// ---- VISUs/StepBlockDetection.TcVIS
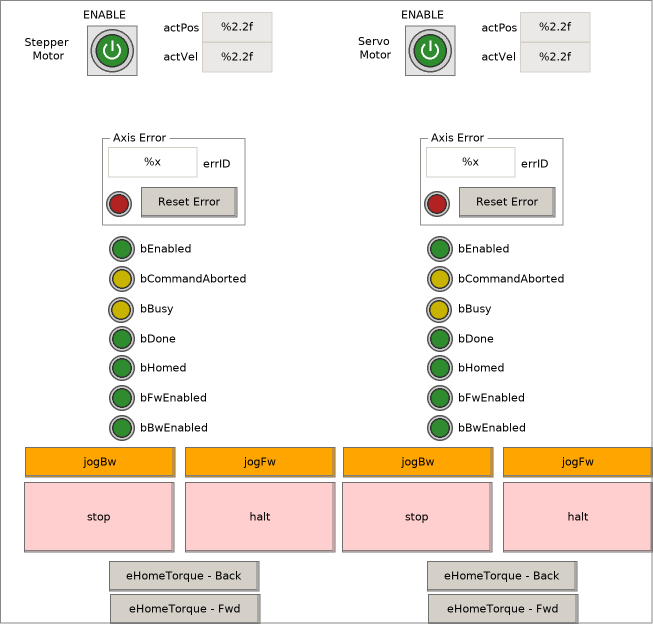
VISUALIZATION StepBlockDetection  // 653x624
    GroupBox (102,130 143x95), "Axis Error"
    Lamp1 (104,189 30x30), variable: GVL.astAxes[1].stStatus.bError, style: Lamp-Lamp1-Red
    Button (141,187 96x30), "Reset Error", pressed state: GVL.astAxes[3].stControl.bReset, text list: 'languageTable', text index: "reset"
        OnMouseClick: toggle GVL.astAxes[1].stControl.bReset
    Textfield (108,147 89x30), "%x", text variable: GVL.astAxes[1].stStatus.nErrorID
    Textfield (200,149 44x30), "errID", text list: 'languageTable', text index: "errID"
    Textfield (137,413 117x30), "bBwEnabled", text list: 'languageTable', text index: "bBwEnabled"
    Lamp1 (107,234 30x30), variable: GVL.astAxes[1].stStatus.bEnabled, style: Lamp-Lamp1-Green
    Textfield (137,234 117x30), "bEnabled", text list: 'languageTable', text index: "bEnabled"
    Lamp1 (107,264 30x30), variable: GVL.astAxes[1].stStatus.bCommandAborted, style: Lamp-Lamp1-Yellow
    Textfield (137,264 117x30), "bCommandAborted", text list: 'languageTable', text index: "bCommandAborted"
    Textfield (137,294 117x30), "bBusy", text list: 'languageTable', text index: "bBusy"
    Lamp1 (107,324 30x30), variable: GVL.astAxes[1].stStatus.bDone, style: Lamp-Lamp1-Green
    Textfield (137,324 117x30), "bDone", text list: 'languageTable', text index: "bDone"
    Lamp1 (107,353 30x30), variable: GVL.astAxes[1].stStatus.bHomed, style: Lamp-Lamp1-Green
    Textfield (137,353 117x30), "bHomed", text list: 'languageTable', text index: "bHomed"
    Lamp1 (107,383 30x30), variable: GVL.astAxes[1].stStatus.bFwEnabled AND NOT GVL.astAxes[1].stStatus.bInterlockedFwd, style: Lamp-Lamp1-Green
    Lamp1 (107,413 30x30), variable: GVL.astAxes[1].stStatus.bBwEnabled AND NOT GVL.astAxes[1].stStatus.bInterlockedBwd, style: Lamp-Lamp1-Green
    Textfield (137,383 117x30), "bFwEnabled", text list: 'languageTable', text index: "bFwEnabled"
    Lamp1 (106,295 30x30), variable: GVL.astAxes[1].stStatus.bBusy, style: Lamp-Lamp1-Yellow
    Textfield (202,12 70x30), "%2.2f", text variable: GVL.astAxes[1].stStatus.fActPosition
    Textfield (148,13 54x30), "actPos", text list: 'languageTable', text index: "actposition"
    Textfield (152,42 49x30), "actVel", text list: 'languageTable', text index: "actVelocity"
    Textfield (202,42 70x30), "%2.2f", text variable: GVL.astAxes[1].stStatus.fActVelocity
    Textfield (80,2 92x26), "ENABLE", text list: 'languageSupport', text index: "enable"
    PowerSwitch (87,24 50x53), variable: GVL.astAxes[1].stControl.bEnable, behaviour: TOGGLE, style: Switch-PowerSwitch-Green
    Button (25,447 150x30), "jogBw", text list: "languageSupport", text index: "jogBw"
        OnMouseDown: execute { GVL.astAxes[1].stControl.eCommand:=E_MotionFunctions.eJog; GVL.astAxes[1].stControl.bJogBwd:= TRUE; }
        OnMouseClick: execute {  }
        OnMouseUp: execute { GVL.astAxes[1].stControl.bJogBwd:= FALSE; }
    Button (185,447 150x30), "jogFw", text list: "languageSupport", text index: "jogFw"
        OnMouseDown: execute { GVL.astAxes[1].stControl.eCommand:=E_MotionFunctions.eJog; GVL.astAxes[1].stControl.bJogFwd:= TRUE; }
        OnMouseClick: execute {  }
        OnMouseUp: execute { GVL.astAxes[1].stControl.bJogFwd:= FALSE; }
    Button (185,482 150x70), "halt", pressed state: GVL.astAxes[1].stControl.bHalt, input disabled if: GVL.astAxes[1].stStatus.bGeared, text list: "languageSupport", text index: "halt"
        toggle GVL.astAxes[1].stControl.bHalt
    Button (24,482 150x70), "stop", pressed state: GVL.astAxes[1].stControl.bStop, input disabled if: GVL.astAxes[1].stStatus.bGeared, text list: "languageSupport", text index: "stop"
        toggle GVL.astAxes[1].stControl.bStop
    Button (109,561 150x30), "eHomeTorque - Back", input disabled if: GVL.astAxes[1].stStatus.bGeared
        OnMouseClick: execute {
            GVL.astAxes[1].stControl.eCommand:=E_MotionFunctions.eHome;
            GVL.astAxes[1].stConfig.eHomeSeq:=E_HomingRoutines.eHomeToBlock_Bwd;
            GVL.astAxes[1].stControl.bExecute:=TRUE;
        }
    Button (110,594 150x30), "eHomeTorque - Fwd", input disabled if: GVL.astAxes[3].stStatus.bGeared
        OnMouseClick: execute {
            GVL.astAxes[1].stControl.eCommand:=E_MotionFunctions.eHome;
            GVL.astAxes[1].stConfig.eHomeSeq:=E_HomingRoutines.eHomeToBlock_Fwd;
            GVL.astAxes[1].stControl.bExecute:=TRUE;
        }
    GroupBox (420,130 143x95), "Axis Error"
    Lamp1 (422,189 30x30), variable: GVL.astAxes[3].stStatus.bError, style: Lamp-Lamp1-Red
    Button (459,187 96x30), "Reset Error", pressed state: GVL.astAxes[3].stControl.bReset, text list: 'languageTable', text index: "reset"
        OnMouseClick: toggle GVL.astAxes[3].stControl.bReset
    Textfield (426,147 89x30), "%x", text variable: GVL.astAxes[3].stStatus.nErrorID
    Textfield (518,149 44x30), "errID", text list: 'languageTable', text index: "errID"
    Textfield (455,413 117x30), "bBwEnabled", text list: 'languageTable', text index: "bBwEnabled"
    Lamp1 (425,234 30x30), variable: GVL.astAxes[3].stStatus.bEnabled, style: Lamp-Lamp1-Green
    Textfield (455,234 117x30), "bEnabled", text list: 'languageTable', text index: "bEnabled"
    Lamp1 (425,264 30x30), variable: GVL.astAxes[3].stStatus.bCommandAborted, style: Lamp-Lamp1-Yellow
    Textfield (455,264 117x30), "bCommandAborted", text list: 'languageTable', text index: "bCommandAborted"
    Textfield (455,294 117x30), "bBusy", text list: 'languageTable', text index: "bBusy"
    Lamp1 (425,324 30x30), variable: GVL.astAxes[3].stStatus.bDone, style: Lamp-Lamp1-Green
    Textfield (455,324 117x30), "bDone", text list: 'languageTable', text index: "bDone"
    Lamp1 (425,353 30x30), variable: GVL.astAxes[3].stStatus.bHomed, style: Lamp-Lamp1-Green
    Textfield (455,353 117x30), "bHomed", text list: 'languageTable', text index: "bHomed"
    Lamp1 (425,383 30x30), variable: GVL.astAxes[3].stStatus.bFwEnabled AND NOT GVL.astAxes[3].stStatus.bInterlockedFwd, style: Lamp-Lamp1-Green
    Lamp1 (425,413 30x30), variable: GVL.astAxes[3].stStatus.bBwEnabled AND NOT GVL.astAxes[3].stStatus.bInterlockedBwd, style: Lamp-Lamp1-Green
    Textfield (455,383 117x30), "bFwEnabled", text list: 'languageTable', text index: "bFwEnabled"
    Lamp1 (424,295 30x30), variable: GVL.astAxes[3].stStatus.bBusy, style: Lamp-Lamp1-Yellow
    Textfield (520,12 70x30), "%2.2f", text variable: GVL.astAxes[3].stStatus.fActPosition
    Textfield (466,13 54x30), "actPos", text list: 'languageTable', text index: "actposition"
    Textfield (470,42 49x30), "actVel", text list: 'languageTable', text index: "actVelocity"
    Textfield (520,42 70x30), "%2.2f", text variable: GVL.astAxes[3].stStatus.fActVelocity
    Textfield (398,2 92x26), "ENABLE", text list: 'languageSupport', text index: "enable"
    PowerSwitch (405,24 50x53), variable: GVL.astAxes[3].stControl.bEnable, behaviour: TOGGLE, style: Switch-PowerSwitch-Green
    Button (343,447 150x30), "jogBw", text list: "languageSupport", text index: "jogBw"
        OnMouseUp: execute { GVL.astAxes[3].stControl.bJogBwd:= FALSE; }
        OnMouseClick: execute {  }
        OnMouseDown: execute { GVL.astAxes[3].stControl.eCommand:=E_MotionFunctions.eJog; GVL.astAxes[3].stControl.bJogBwd:= TRUE; }
    Button (503,447 150x30), "jogFw", text list: "languageSupport", text index: "jogFw"
        OnMouseUp: execute { GVL.astAxes[3].stControl.bJogFwd:= FALSE; }
        OnMouseClick: execute {  }
        OnMouseDown: execute { GVL.astAxes[3].stControl.eCommand:=E_MotionFunctions.eJog; GVL.astAxes[3].stControl.bJogFwd:= TRUE; }
    Button (503,482 150x70), "halt", pressed state: GVL.astAxes[3].stControl.bHalt, input disabled if: GVL.astAxes[3].stStatus.bGeared, text list: "languageSupport", text index: "halt"
        toggle GVL.astAxes[3].stControl.bHalt
    Button (342,482 150x70), "stop", pressed state: GVL.astAxes[3].stControl.bStop, input disabled if: GVL.astAxes[3].stStatus.bGeared, text list: "languageSupport", text index: "stop"
        toggle GVL.astAxes[3].stControl.bStop
    Button (427,561 150x30), "eHomeTorque - Back", input disabled if: GVL.astAxes[3].stStatus.bGeared
        OnMouseClick: execute {
            GVL.astAxes[3].stControl.eCommand:=E_MotionFunctions.eHome;
            GVL.astAxes[3].stConfig.eHomeSeq:=E_HomingRoutines.eHomeToBlock_Bwd;
            GVL.astAxes[3].stControl.bExecute:=TRUE;
        }
    Button (428,594 150x30), "eHomeTorque - Fwd", input disabled if: GVL.astAxes[3].stStatus.bGeared
        OnMouseClick: execute {
            GVL.astAxes[3].stControl.eCommand:=E_MotionFunctions.eHome;
            GVL.astAxes[3].stConfig.eHomeSeq:=E_HomingRoutines.eHomeToBlock_Fwd;
            GVL.astAxes[3].stControl.bExecute:=TRUE;
        }
    Label (5,34 87x30), "Stepper Motor"
    Label (332,33 87x30), "Servo Motor"
END_VISUALIZATION
